// TIA Portal V15.1 export
// export: Created 2024-06-21T08:41:08.1695515Z, ExportSetting WithDefaults, DisplayName Totally Integrated Automation Portal, DisplayVersion V15.1 Update 5, DisplayName TIA Portal Openness, DisplayVersion V15.1 Update 5, DisplayName SINAMICS Startdrive Advanced, DisplayVersion V15.1, DisplayName G130, G150, S120, S150, SINAMICS MV, S210, DisplayVersion V15.1, DisplayName G110M, G120, G120C, G120D, G120P, DisplayVersion V15.1, DisplayName STEP 7 Professional, DisplayVersion V15.1 Update 5, DisplayName STEP 7 Safety, DisplayVersion V15.1, DisplayName WinCC Professional, DisplayVersion V15.1 Update 5, DisplayName SIMATIC Visualization Architect, DisplayVersion V15.1
FUNCTION_BLOCK "LGBLineFeedSub"   // FB6707, SCL
{ S7_Optimized_Access := 'TRUE' }
AUTHOR : VCG
FAMILY : Conv
VERSION : 0.1
// stored: AutoNumber false, IsIECCheckEnabled false, IsRetainMemResEnabled false, MemoryReserve 100, SetENOAutomatically False, UDAEnableTagReadback false
   VAR_INPUT
      I_BodyPresent { ExternalAccessible := 'False'; ExternalVisible := 'False'; ExternalWritable := 'False'} : Bool;   // Body present, ready for infeed begin
      I_GapsAllowed { ExternalAccessible := 'False'; ExternalVisible := 'False'; ExternalWritable := 'False'} : Bool;   // Gaps allowed
      I_InfdWaitCond { ExternalAccessible := 'False'; ExternalVisible := 'False'; ExternalWritable := 'False'} : Bool;   // Infeed wait - Condition
      I_InfdWaitDoneCond { ExternalAccessible := 'False'; ExternalVisible := 'False'; ExternalWritable := 'False'} : Bool;   // Infeed wait - Condition done
      I_OutfdWaitCond { ExternalAccessible := 'False'; ExternalVisible := 'False'; ExternalWritable := 'False'} : Bool;   // Outfeed wait - Condition
      I_OutfdWaitDoneCond { ExternalAccessible := 'False'; ExternalVisible := 'False'; ExternalWritable := 'False'} : Bool;   // Outfeed wait - Condition done
   END_VAR
   VAR_OUTPUT
      O_InfdBegin { ExternalAccessible := 'False'; ExternalVisible := 'False'; ExternalWritable := 'False'} : Bool;   // Infeed begin (to conveyor module)
      O_StopReqInfdWait { ExternalAccessible := 'False'; ExternalVisible := 'False'; ExternalWritable := 'False'} : Bool;   // Stop request from infeed wait
      O_StopReqOutfdWait { ExternalAccessible := 'False'; ExternalVisible := 'False'; ExternalWritable := 'False'} : Bool;   // Stop request from outfeed wait
      O_PartsAtFixedLineStop { ExternalAccessible := 'False'; ExternalVisible := 'False'; ExternalWritable := 'False'} : Bool;   // Parts are at fixed line stop position
      O_AlarmNoBodyPresent { ExternalAccessible := 'False'; ExternalVisible := 'False'; ExternalWritable := 'False'} : Bool;   // It's time for INFEED BEGIN but there is now body in position
   END_VAR
   VAR_IN_OUT
      IO_ShiftRegData : "ShiftRegData";   // Line data- from shiftregister
      H_HMI : "H_HMI";   // Animation
      H_GBLineFeed : "H_GBLineFeed";   // Animation
      C_Config : "LineFeedConfig";   // Config
   END_VAR
   VAR
      AlarmNoBodyPresent { ExternalAccessible := 'False'; ExternalVisible := 'False'; ExternalWritable := 'False'} : Bool;   // It's time for INFEED BEGIN but there is no body in position
      i { ExternalAccessible := 'False'; ExternalVisible := 'False'; ExternalWritable := 'False'} : Int;   // Index
      ZoneFLSFirstPos { ExternalAccessible := 'False'; ExternalVisible := 'False'; ExternalWritable := 'False'} : Int;   // First fixed line stop zone
      ZoneFLSLastPos { ExternalAccessible := 'False'; ExternalVisible := 'False'; ExternalWritable := 'False'} : Int;   // Last fixed line stop zone
      BodyPitchCorr { ExternalAccessible := 'False'; ExternalVisible := 'False'; ExternalWritable := 'False'} : Int;   // Bodypitch correction value (cm)
      InfdBegin { ExternalAccessible := 'False'; ExternalVisible := 'False'; ExternalWritable := 'False'} : Bool;   // Infeed begin
      StopReqInfdWait { ExternalAccessible := 'False'; ExternalVisible := 'False'; ExternalWritable := 'False'} : Bool;   // Stop request Infeed wait
      StopReqInfdWaitCond { ExternalAccessible := 'False'; ExternalVisible := 'False'; ExternalWritable := 'False'} : Bool;   // Stop request Infeed wait - Condition
      StopReqOutfdWait { ExternalAccessible := 'False'; ExternalVisible := 'False'; ExternalWritable := 'False'} : Bool;   // Stop request Outfeed wait
      StopReqOutfdWaitCond { ExternalAccessible := 'False'; ExternalVisible := 'False'; ExternalWritable := 'False'} : Bool;   // Stop request Outfeed wait - Condition
      PartAtFLS { ExternalAccessible := 'False'; ExternalVisible := 'False'; ExternalWritable := 'False'} : Bool;   // Parts are at fixed line stop position
      PartAtFLSSet { ExternalAccessible := 'False'; ExternalVisible := 'False'; ExternalWritable := 'False'} : Bool;   // Parts are at fixed line stop position
      PartAtFLSRes { ExternalAccessible := 'False'; ExternalVisible := 'False'; ExternalWritable := 'False'} : Bool;   // Parts are at fixed line stop position
      R_TRIG_StopReqInfdWaitCond { ExternalAccessible := 'False'; ExternalVisible := 'False'; ExternalWritable := 'False'} : R_TRIG;   // TRIGGER
      R_TRIG_StopReqOutfdWaitCond { ExternalAccessible := 'False'; ExternalVisible := 'False'; ExternalWritable := 'False'} : R_TRIG;   // TRIGGER
      T_InfBegin { ExternalAccessible := 'False'; ExternalVisible := 'False'; ExternalWritable := 'False'} : TOF_TIME;   // TIMER
   END_VAR
   VAR_TEMP
      HMICMD : Struct   // Temp
         Spare0 : Bool;   // Spare
         Spare1 : Bool;   // Spare
         Spare2 : Bool;   // Spare
         Spare3 : Bool;   // Spare
         Spare4 : Bool;   // Spare
         Spare5 : Bool;   // Spare
         Spare6 : Bool;   // Spare
         Spare7 : Bool;   // Spare
         Spare8 : Bool;   // Spare
         Spare9 : Bool;   // Spare
         Spare10 : Bool;   // Spare
         Spare11 : Bool;   // Spare
         Spare12 : Bool;   // Spare
         Spare13 : Bool;   // Spare
         Spare14 : Bool;   // Spare
         Spare15 : Bool;   // Spare
         Spare16 : Bool;   // Spare
         Spare17 : Bool;   // Spare
         Spare18 : Bool;   // Spare
         Spare19 : Bool;   // Spare
         Spare20 : Bool;   // Spare
         Spare21 : Bool;   // Spare
         Spare22 : Bool;   // Spare
         Spare23 : Bool;   // Spare
         Spare24 : Bool;   // Spare
         Spare25 : Bool;   // Spare
         Spare26 : Bool;   // Spare
         Spare27 : Bool;   // Spare
         Spare28 : Bool;   // Spare
         Spare29 : Bool;   // Spare
         Spare30 : Bool;   // Spare
         Spare31 : Bool;   // Spare
      END_STRUCT;
   END_VAR
BEGIN
   REGION *** HMI Commands ***
       "LDWordToBit"(I_DWord := #H_GBLineFeed.H_HMICmd,
                     O_0 => #HMICMD.Spare0,
                     O_1 => #HMICMD.Spare1,
                     O_2 => #HMICMD.Spare2,
                     O_3 => #HMICMD.Spare3,
                     O_4 => #HMICMD.Spare4,
                     O_5 => #HMICMD.Spare5,
                     O_6 => #HMICMD.Spare6,
                     O_7 => #HMICMD.Spare7,
                     O_8 => #HMICMD.Spare8,
                     O_9 => #HMICMD.Spare9,
                     O_10 => #HMICMD.Spare10,
                     O_11 => #HMICMD.Spare11,
                     O_12 => #HMICMD.Spare12,
                     O_13 => #HMICMD.Spare13,
                     O_14 => #HMICMD.Spare14,
                     O_15 => #HMICMD.Spare15,
                     O_16 => #HMICMD.Spare16,
                     O_17 => #HMICMD.Spare17,
                     O_18 => #HMICMD.Spare18,
                     O_19 => #HMICMD.Spare18,
                     O_20 => #HMICMD.Spare19,
                     O_21 => #HMICMD.Spare21,
                     O_22 => #HMICMD.Spare22,
                     O_23 => #HMICMD.Spare23,
                     O_24 => #HMICMD.Spare24,
                     O_25 => #HMICMD.Spare25,
                     O_26 => #HMICMD.Spare26,
                     O_27 => #HMICMD.Spare27,
                     O_28 => #HMICMD.Spare28,
                     O_29 => #HMICMD.Spare29,
                     O_30 => #HMICMD.Spare30,
                     O_31 => #HMICMD.Spare31);

       // Body Pitch correction (Infeed Begin)
       #BodyPitchCorr := #H_GBLineFeed.H_BodyPitchCorr;

   END_REGION

   REGION *** INIT ***

       #ZoneFLSFirstPos := 1;
       #ZoneFLSLastPos := #IO_ShiftRegData.NbrOfWorkZones;

   END_REGION

   REGION *** Alarms ***

       //It's time for INFEED BEGIN but there is now body in position
       IF (#InfdBegin AND NOT #I_BodyPresent AND NOT #I_GapsAllowed AND NOT #IO_ShiftRegData.LineIsEmpty AND #C_Config.EnableAlarmNoBodyPresent) THEN
           #AlarmNoBodyPresent := True;
       END_IF;

       IF (#I_BodyPresent OR #I_GapsAllowed OR #IO_ShiftRegData.LineIsEmpty OR NOT #C_Config.EnableAlarmNoBodyPresent) THEN
           #AlarmNoBodyPresent := False;
       END_IF;

   END_REGION

   REGION *** Parts at 'Fixed Line Stop' ***

       #i := 0;
       #PartAtFLS := False;
       WHILE #IO_ShiftRegData.Zone[#i].TagID = 0 AND #i <= #ZoneFLSLastPos DO
           #i := #i + 1;
       END_WHILE;
       IF (#i >= 0) AND (#i <= #ZoneFLSLastPos) THEN
           #PartAtFLSSet := (#IO_ShiftRegData.Zone[#i].ActualPosition - #IO_ShiftRegData.Zone[#i].StartPosition >= 0) AND ((#IO_ShiftRegData.Zone[#i].ActualPosition - #IO_ShiftRegData.Zone[#i].StartPosition) <= (#C_Config.WindowDist / 2));
           #PartAtFLSRes := (#IO_ShiftRegData.Zone[#i].EndPosition - #IO_ShiftRegData.Zone[#i].ActualPosition > 0) AND ((#IO_ShiftRegData.Zone[#i].EndPosition - #IO_ShiftRegData.Zone[#i].ActualPosition) <= #C_Config.RampDownDist);
           #PartAtFLS := #PartAtFLSRes OR #PartAtFLSSet;
       END_IF;

   END_REGION

   REGION *** Infeed Begin ***

       IF #IO_ShiftRegData.SetpointBodyPitch > 0 THEN
           IF #IO_ShiftRegData.LineIsEmpty THEN
               #InfdBegin := True;
           ELSIF NOT #IO_ShiftRegData.LineIsEmpty AND NOT #C_Config.BodyPitchMinDistance THEN
               #InfdBegin := (#IO_ShiftRegData.ActualBodyPitchZoneX >= INT_TO_REAL(#IO_ShiftRegData.SetpointBodyPitch + #BodyPitchCorr)) AND (#IO_ShiftRegData.ActualBodyPitchZoneX <= INT_TO_REAL(#IO_ShiftRegData.SetpointBodyPitch + #BodyPitchCorr + #C_Config.WindowDist));
           ELSIF NOT #IO_ShiftRegData.LineIsEmpty AND #C_Config.BodyPitchMinDistance THEN
               #InfdBegin := (#IO_ShiftRegData.ActualBodyPitch >= INT_TO_REAL(#IO_ShiftRegData.SetpointBodyPitch + #BodyPitchCorr));
           END_IF;
       END_IF;

   END_REGION

   REGION *** Stop request - Infeed wait ***

       #StopReqInfdWaitCond := #I_InfdWaitCond AND NOT #I_GapsAllowed AND #PartAtFLS;

       #R_TRIG_StopReqInfdWaitCond(CLK := #StopReqInfdWaitCond);

       IF #R_TRIG_StopReqInfdWaitCond.Q THEN
           #StopReqInfdWait := True;
       END_IF;

       IF #I_InfdWaitDoneCond OR #I_GapsAllowed THEN
           #StopReqInfdWait := FALSE;
       END_IF;

   END_REGION

   REGION *** Stop request - Outfeed wait ***

       #StopReqOutfdWaitCond := #I_OutfdWaitCond AND #PartAtFLS;

       #R_TRIG_StopReqOutfdWaitCond(CLK := #StopReqOutfdWaitCond);

       IF #R_TRIG_StopReqOutfdWaitCond.Q THEN
           #StopReqOutfdWait := TRUE;
       END_IF;

       IF #I_OutfdWaitDoneCond THEN
           #StopReqOutfdWait := FALSE;
       END_IF;

   END_REGION

   REGION *** Outputs ***

       #O_InfdBegin := #InfdBegin;
       #O_StopReqInfdWait := #StopReqInfdWait;
       #O_StopReqOutfdWait := #StopReqOutfdWait;
       #O_PartsAtFixedLineStop := #PartAtFLS;
       #O_AlarmNoBodyPresent := #AlarmNoBodyPresent;

   END_REGION

   REGION *** HMI ***

       REGION *** Values ***
           #H_GBLineFeed.H_BodyPitch := #IO_ShiftRegData.SetpointBodyPitch;
           #H_HMI.H_IAnim3 := #IO_ShiftRegData.SetpointBodyPitch;

           #H_GBLineFeed.H_BodyPitchAct := REAL_TO_INT(#IO_ShiftRegData.ActualBodyPitch);
           #H_HMI.H_IAnim2 := REAL_TO_DINT(#IO_ShiftRegData.ActualBodyPitch);

           IF REAL_TO_INT(#IO_ShiftRegData.ActualBodyPitch) >= #IO_ShiftRegData.SetpointBodyPitch THEN
               #H_GBLineFeed.H_BodyPitchAct := REAL_TO_INT(#IO_ShiftRegData.ActualBodyPitch) - #IO_ShiftRegData.SetpointBodyPitch;
               #H_HMI.H_IAnim2 := REAL_TO_INT(#IO_ShiftRegData.ActualBodyPitch) - #IO_ShiftRegData.SetpointBodyPitch;
               IF #H_GBLineFeed.H_BodyPitchAct >= #IO_ShiftRegData.SetpointBodyPitch THEN
                   #H_GBLineFeed.H_BodyPitchAct := #IO_ShiftRegData.SetpointBodyPitch;
                   #H_HMI.H_IAnim2 := #IO_ShiftRegData.SetpointBodyPitch;
               END_IF;
           END_IF;

           //Partnumber and position Shift Register
           #H_GBLineFeed.H_ShiftRegDataZoneA_TagID := #IO_ShiftRegData.Zone[0].TagID;
           #H_GBLineFeed.H_ShiftRegDataZoneA_Position := REAL_TO_DINT(#IO_ShiftRegData.Zone[0].ActualPosition);
           #H_GBLineFeed.H_ShiftRegDataZoneB_TagID := #IO_ShiftRegData.Zone[1].TagID;
           #H_GBLineFeed.H_ShiftRegDataZoneB_Position := REAL_TO_DINT(#IO_ShiftRegData.Zone[1].ActualPosition);

           #H_GBLineFeed.H_ShiftRegDataZoneY_TagID := #IO_ShiftRegData.Zone[#ZoneFLSLastPos].TagID;
           #H_GBLineFeed.H_ShiftRegDataZoneY_Position := REAL_TO_DINT(#IO_ShiftRegData.Zone[#ZoneFLSLastPos].ActualPosition);
           #H_GBLineFeed.H_ShiftRegDataZoneZ_TagID := #IO_ShiftRegData.Zone[#ZoneFLSLastPos + 1].TagID;
           #H_GBLineFeed.H_ShiftRegDataZoneZ_Position := REAL_TO_DINT(#IO_ShiftRegData.Zone[#ZoneFLSLastPos + 1].ActualPosition);

       END_REGION

       REGION *** Animations ***

           #T_InfBegin(IN:= #InfdBegin,
                     PT:= T#2s,
                     Q=> "NotUsedBool",
                     ET=> "NotUsedDInt");

                     "LBitToDword"(I_0 := #T_InfBegin.Q,
                         I_1 := FALSE,
                         I_2 := FALSE,
                         I_3 := #PartAtFLS,
                         I_4 := FALSE,
                         I_5 := FALSE,
                         I_6 := FALSE,
                         I_7 := FALSE,
                         I_8 := FALSE,
                         I_9 := FALSE,
                         I_10 := FALSE,
                         I_11 := FALSE,
                         I_12 := FALSE,
                         I_13 := FALSE,
                         I_14 := FALSE,
                         I_15 := FALSE,
                         I_16 := FALSE,
                         I_17 := FALSE,
                         I_18 := FALSE,
                         I_19 := FALSE,
                         I_20 := FALSE,
                         I_21 := FALSE,
                         I_22 := FALSE,
                         I_23 := FALSE,
                         I_24 := FALSE,
                         I_25 := FALSE,
                         I_26 := FALSE,
                         I_27 := FALSE,
                         I_28 := FALSE,
                         I_29 := FALSE,
                         I_30 := FALSE,
                         I_31 := FALSE,
                         O_DWord => #H_GBLineFeed.H_Anim[1].H_DWord);

       END_REGION

       REGION *** Icon Animation ***

           "LIAnimDWord"(I_SetPos := FALSE,
                         I_ResetPos := FALSE,
                         I_Active := #T_InfBegin.Q,
                         I_Visible := FALSE,
                         I_OutOfUse := FALSE,
                         I_IntlkSet := FALSE,
                         I_IntlkReset := FALSE,
                         I_IntlkSetAlm := FALSE,
                         I_IntlkResetAlm := FALSE,
                         I_ManualMode := FALSE,
                         I_FncSelInHMI := FALSE,
                         I_AnySelected := FALSE,
                         I_AlarmA := FALSE,
                         I_AlarmB := FALSE,
                         I_AlarmC := FALSE,
                         I_AlarmD := FALSE,
                         I_SafetyOk := FALSE,
                         I_Service := TRUE,
                         I_Spare1 := FALSE,
                         I_Spare2 := FALSE,
                         I_Spare3 := FALSE,
                         I_Spare4 := FALSE,
                         I_Spare5 := FALSE,
                         I_Spare6 := FALSE,
                         I_Spare7 := FALSE,
                         I_Spare8 := FALSE,
                         I_Spare9 := FALSE,
                         I_Spare10 := FALSE,
                         I_Spare11 := FALSE,
                         I_Spare12 := FALSE,
                         I_Spare13 := FALSE,
                         I_Spare14 := FALSE,
                         H_IAnim => #H_HMI.H_IAnim);

       END_REGION

   END_REGION
END_FUNCTION_BLOCK
